// TIA Portal V20 export
ORGANIZATION_BLOCK "CFC_Cyclic interrupt_5"   // OB1035, CFC, CyclicInterrupt
{ S7_Optimized_Access := 'TRUE' }
AUTHOR : CFC
FAMILY : CFCPlus
VERSION : 1.0
// stored: AutoNumber false
   VAR_INPUT
      Initial_Call : Bool;   // Initial call of this OB
      Event_Count : Int;   // Events discarded
   END_VAR
   VAR_TEMP
      t_out : UInt;
   END_VAR
BEGIN
END_ORGANIZATION_BLOCK
